FUNCTION_BLOCK App4_ReactorLevel (* Composite Function Block Type *)
  (* Standard: 61499-2 *)
  (* Version 0.0, 2018-11-06, 4DIAC-IDE, 4DIAC-Consortium *)
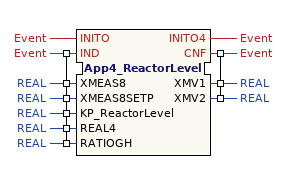
  EVENT_INPUT
    INITO; (* Initialization Request *)
    IND WITH XMEAS8, XMEAS8SETP, KP_ReactorLevel, REAL4, RATIOGH; (* Normal Execution Request *)
  END_EVENT
  EVENT_OUTPUT
    INITO4; (* Initialization Confirm *)
    CNF WITH XMV1, XMV2; (* Execution Confirmation *)
  END_EVENT
  VAR_INPUT
    XMEAS8 : REAL;
    XMEAS8SETP : REAL;
    KP_ReactorLevel : REAL;
    REAL4 : REAL;
    RATIOGH : REAL;
  END_VAR
  VAR_OUTPUT
    XMV1 : REAL;
    XMV2 : REAL;
  END_VAR
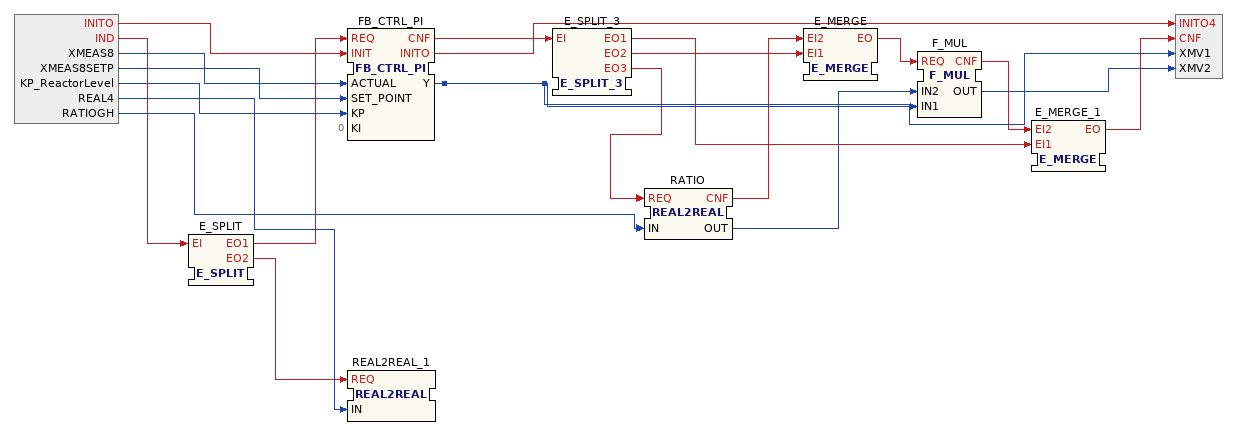
  FBS
    E_SPLIT : E_SPLIT;
    E_MERGE : E_MERGE;
    RATIO : REAL2REAL;
    F_MUL : F_MUL;
    FB_CTRL_PI : FB_CTRL_PI(KI := 0);
    REAL2REAL_1 : REAL2REAL;
    E_SPLIT_3 : E_SPLIT_3;
    E_MERGE_1 : E_MERGE;
  END_FBS
  EVENT_CONNECTIONS
    E_SPLIT.EO1 TO FB_CTRL_PI.REQ;
    E_SPLIT.EO2 TO REAL2REAL_1.REQ;
    IND TO E_SPLIT.EI;
    RATIO.CNF TO E_MERGE.EI2;
    E_MERGE.EO TO F_MUL.REQ;
    FB_CTRL_PI.CNF TO E_SPLIT_3.EI;
    F_MUL.CNF TO E_MERGE_1.EI2;
    E_SPLIT_3.EO1 TO E_MERGE_1.EI1;
    E_SPLIT_3.EO2 TO E_MERGE.EI1;
    E_SPLIT_3.EO3 TO RATIO.REQ;
    E_MERGE_1.EO TO CNF;
    INITO TO FB_CTRL_PI.INIT;
    FB_CTRL_PI.INITO TO INITO4;
  END_CONNECTIONS
  DATA_CONNECTIONS
    RATIO.OUT TO F_MUL.IN2;
    FB_CTRL_PI.Y TO F_MUL.IN1;
    FB_CTRL_PI.Y TO XMV1;
    F_MUL.OUT TO XMV2;
    XMEAS8 TO FB_CTRL_PI.ACTUAL;
    XMEAS8SETP TO FB_CTRL_PI.SET_POINT;
    KP_ReactorLevel TO FB_CTRL_PI.KP;
    REAL4 TO REAL2REAL_1.IN;
    RATIOGH TO RATIO.IN;
  END_CONNECTIONS
END_FUNCTION_BLOCK
